// TIA Portal V20 export
DATA_BLOCK "DB_ReadDateAndTime"   // DB9
// stored: InstanceOfName FB_ReadDateAndTime, InstanceOfType FB
"FB_ReadDateAndTime"
   // VAR
   //    sDateAndTime : DTL;
   //    sCurrentDT : Struct
   //       sYear : UInt;
   //       sMonth : USInt;
   //       sDay : USInt;
   //       sHour : USInt;
   //       sMinute : USInt;
   //       sSecond : USInt;
   //       sNanoSecond : UDInt;
   //    END_STRUCT;
   // END_VAR
BEGIN
END_DATA_BLOCK
